// TIA Portal V20 export
// export: Created 2025-12-01T14:56:19.2822619Z, ExportSetting None, DisplayName Totally Integrated Automation Portal, DisplayVersion V20 Update 3, DisplayName TIA Portal Openness, DisplayVersion V20 Update 3, DisplayName TIA Portal Version Control Interface, DisplayVersion V20 Update 3, DisplayName STEP 7 Professional, DisplayVersion V20 Update 3, DisplayName STEP 7 Safety, DisplayVersion V20 Update 2, DisplayName WinCC Basic/Comfort/Advanced, DisplayVersion V20 Update 3, DisplayName WinCC Professional, DisplayVersion V20 Update 3, DisplayName WinCC Unified, DisplayVersion V20 Update 3
TYPE "Registro"
   STRUCT
      T_Etapa_Cargada : Time;   // Tiempo en Etapa Cargada
      T_Etapa_Carga_E0 : Time;
      T_Etapa_Carga_E1 : Time;   // Tiempo Carga por E1
      T_Etapa_Carga_E2 : Time;   // Tiempo Carga por E2
      T_Etapa_Carga_E3 : Time;   // Tiempo Carga por E3
      T_Etapa_Carga_E4 : Time;   // Tiempo Carga por E4
      T_Etapa_Descarga_S0 : Time;
      T_Etapa_Descarga_S1 : Time;   // Tiempo Descarga por S1
      T_Etapa_Descarga_S2 : Time;   // Tiempo Descarga por S2
      T_Etapa_Descarga_S3 : Time;   // Tiempo Descarga por S3
      T_Etapa_Descarga_S4 : Time;   // Tiempo Descarga por S4
      T_Rodillos : Time;   // Tiempo movimiento de Rodillos
      T_Cadenas : Time;   // Tiempo movimiento de Cadenas
      T_Giro : Time;   // Tiempo movimiento de Giro
      T_Subir_Transfer : Time;   // Tiempo movimiento de Subida Transfer
      T_Bajar_Transfer : Time;   // Tiempo movimiento de Bajada Transfer
      T_Total : Time;
   END_STRUCT;
END_TYPE
